FUNCTION_BLOCK LinearServoNC EXTENDS FBA_TrifectaDrive IMPLEMENTS I_EncodedDrive
VAR_INPUT
	bEnable : BOOL;
END_VAR
VAR_OUTPUT	
	ready : BOOL;
	position : LREAL;
	velocity : LREAL;
END_VAR
VAR
	servo : ServoNC;
	home AT %I* : BOOL;
	extendLimit AT %I* : BOOL;
	retractLimit AT %I* : BOOL;
END_VAR
VAR_STAT CONSTANT
	targetingVelocity : INT := 500;
	continuousVelocity : INT := 100;
END_VAR

override();

servo(bEnable:= bEnable, ready=> , position=> , velocity=> );

ready := bEnable AND NOT Active AND HomeSet;

PROPERTY Active : BOOL
GET
Active := servo.Active;
END_GET
END_PROPERTY

PROPERTY CurrentPosition : LREAL
GET
CurrentPosition := position;
END_GET
END_PROPERTY

PROPERTY Error : BOOL
GET
error := servo.Error;
END_GET
END_PROPERTY

METHOD homingSequence : BOOL
(*
homing sequence is different for linear motion devices with limit sensors
*)
CASE step OF
	Homing.IDLE:
		reset();
		IF bEnable THEN
			step := Homing.START;
		END_IF
		
	Homing.START:
		IF AtHome THEN
			stop();
			
		ELSIF AtInnerLimit THEN
			step := Homing.RETRY;
			
		ELSE
			moveContinuous(direction:= MC_Positive_Direction);
		END_IF
		
	Homing.RETRY:
		IF AtOuterLimit THEN
			moveContinuous(direction:= MC_Positive_Direction);
		ELSE
			moveContinuous(direction:= MC_Negative_Direction);
		END_IF
		
	Homing.STOP:
		IF velocity = 0 THEN
			step := Homing.SET;
		ELSE
			stop();
		END_IF
		
	Homing.SET:
		IF position = 0 THEN
			step := Homing.DONE;
		ELSE
			setPosition(newPosition:= 0);
		END_IF
		
	Homing.DONE:
		homingComplete := TRUE;
		step := Homing.IDLE;
		
END_CASE
END_METHOD

METHOD moveAbsolute : BOOL
VAR_INPUT
	newTarget : LREAL;
END_VAR
(*
VAR_OUTPUT
	fault : BOOL;
END_VAR
*)
servo.moveAbsolute(newTarget:= newTarget);

moveAbsolute := servo.CurrentPosition = newTarget;
END_METHOD

METHOD moveContinuous : BOOL
VAR_INPUT
	//direction : BOOL; //direction (F = inwards, T = outwards)
	direction : MC_Direction;
END_VAR
servo.moveContinuous(direction:= direction);
END_METHOD

METHOD moveRelative : BOOL
VAR_INPUT
	distance : LREAL;
END_VAR
servo.moveRelative(distance:= distance);
END_METHOD

METHOD PRIVATE override : BOOL
VAR_INPUT
END_VAR
(*
-at home and attempting to traverse outward
-at outer limit and attempting to traverse outward
-at inner limit and attempting to traverse inwards
*)
(*
inward = negative direction, negative velocity
outward = positive direction, positive velocity
*)

IF error THEN
	stop();
	reset();
	
ELSIF
	(NOT enableDualSideTraverse AND AtHome AND (TargetPosition > CurrentPosition OR velocity > 0)) OR
	(AtInnerLimit AND (TargetPosition > CurrentPosition OR velocity > 0)) OR
	(AtOuterLimit AND (TargetPosition < CurrentPosition OR velocity < 0))
THEN
	stop();
END_IF
END_METHOD

METHOD reset : BOOL
VAR_INPUT
END_VAR
reset := servo.reset();
END_METHOD

METHOD setPosition : BOOL
VAR_INPUT
	newPosition : LREAL;
END_VAR
servo.setPosition(newPosition:= newPosition);
END_METHOD

METHOD stop : BOOL
VAR_INPUT
END_VAR
servo.stop();
END_METHOD

PROPERTY TargetPosition : LREAL
GET
END_GET
END_PROPERTY

METHOD toHome : BOOL
VAR_INPUT
END_VAR
servo.toHome();
END_METHOD

END_FUNCTION_BLOCK

(* stored: Version 1.1.0.1, ProductVersion 3.1.4024.11
   POU LinearServoNC: Id {6a71c24b-e121-4635-9ee8-54e86420da1c}, SpecialFunc None
   Folder Private: Id {6469a0cb-b276-4ed0-9c96-660d2cb3cb01}
   Folder Properties: Id {2c72d08d-a3d9-44fe-a49e-fde63c7b6d42}
   Property Active: Id {42c3c90f-8aef-4b8a-a8da-29af834cfb45}
   Get Get: Id {bc64cf50-6f57-4b35-b0c3-c8dc52548241}
   Property CurrentPosition: Id {84239ffc-cf90-4509-971e-2670c4b7c146}
   Get Get: Id {d9683bb0-3645-4356-878c-5a2e47a29b8a}
   Property Error: Id {a4e2a042-d51c-4124-afa7-310d6c9b2ccb}
   Get Get: Id {1a2c45b2-9a87-4add-a5f6-66c0f5c16aa9}
   Method homingSequence: Id {42a6228d-3424-4599-956f-2e24eab209bc}
   Method moveAbsolute: Id {8b6b09ff-4944-4076-87ac-211681c4fd5c}
   Method moveContinuous: Id {1b42a1d1-5780-4556-a8a9-8bdd18b8065f}
   Method moveRelative: Id {fefd542d-684b-455c-8676-f10bc0192545}
   Method override: Id {7f0c1445-2dad-41af-a5d4-699b45d88d4c}
   Method reset: Id {19da08b7-85d2-4185-8ac0-74ccd63de424}
   Method setPosition: Id {5ee3c031-8bdb-416b-9e14-f1453cfee97e}
   Method stop: Id {272d864d-02a5-46e4-8492-3b483738d97a}
   Property TargetPosition: Id {b1b94a76-ff8e-442c-9aae-50c9bffe232c}
   Get Get: Id {9c471c4d-ee95-46be-80e3-d7bc7c3a9200}
   Method toHome: Id {6ef6dea7-91dd-4001-b34e-5cd42de9cb8c} *)
